FUNCTION_BLOCK OP_Select_Str (* Basic Function Block Type *)
  (* Standard: 61499-2 *)
  (* Version 0.0, 4/16/2020, prana, nxtControl GmbH, Template *)
  PACKAGE Main;
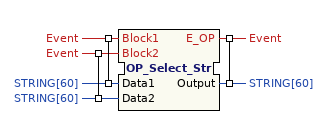
  EVENT_INPUT
    Block1 WITH Data1; (* Initialization Request *)
    Block2 WITH Data2; (* Normal Execution Request *)
  END_EVENT
  EVENT_OUTPUT
    E_OP WITH Output; (* Initialization Confirm *)
  END_EVENT
  VAR_INPUT
    Data1 : STRING[60]; (* Input event qualifier *)
    Data2 : STRING[60];
  END_VAR
  VAR_OUTPUT
    Output : STRING[60]; (* Output event qualifier *)
  END_VAR
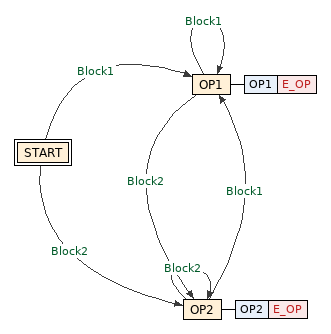
  EC_STATES
    START; (* Initial State *)
    OP1 : OP1 -> E_OP; (* Initialization *)
    OP2 : OP2 -> E_OP; (* Normal execution *)
  END_STATES
  EC_TRANSITIONS
    START TO OP1 := Block1;
    START TO OP2 := Block2;
    OP2 TO OP1 := Block1;
    OP1 TO OP2 := Block2;
    OP1 TO OP1 := Block1;
    OP2 TO OP2 := Block2;
  END_TRANSITIONS
  ALGORITHM OP1 IN ST: (* Initialization algorithm *)
Output := Data1 ;
Block1 := FALSE;
  END_ALGORITHM
  ALGORITHM OP2 IN ST:
Output := Data2;
Block2 := FALSE;
  END_ALGORITHM
END_FUNCTION_BLOCK
